// TIA Portal V20 export
// export: Created 2025-12-01T14:56:18.2640072Z, ExportSetting None, DisplayName Totally Integrated Automation Portal, DisplayVersion V20 Update 3, DisplayName TIA Portal Openness, DisplayVersion V20 Update 3, DisplayName TIA Portal Version Control Interface, DisplayVersion V20 Update 3, DisplayName STEP 7 Professional, DisplayVersion V20 Update 3, DisplayName STEP 7 Safety, DisplayVersion V20 Update 2, DisplayName WinCC Basic/Comfort/Advanced, DisplayVersion V20 Update 3, DisplayName WinCC Professional, DisplayVersion V20 Update 3, DisplayName WinCC Unified, DisplayVersion V20 Update 3
TYPE "UDT_VarLenze"
   STRUCT
      VF_Aviso : Bool;
      VF_Problema : Bool;
      VF01_EnAvance : Bool;
      VF01_EnRetroceso : Bool;
      VF02_EnAvance : Bool;
      VF02_EnRetroceso : Bool;
      VF01_Orden : Bool;
      VF02_Orden : Bool;
      VF_Ready : Bool;
      VF_SpeedCero : Bool;
      VF_NodoPresente : Bool;
      Bit_13 : Bool;
      Bit_14 : Bool;
      Bit_15 : Bool;
      Bit_16 : Bool;
      VF_SalidaDigital : Bool;
      ConsignaReal : Int;
      ConsignaReal_TMP : DInt;
      TIMConMutacion : UDInt;   // Temporizador de ConMutación de los Motores
   END_STRUCT;
END_TYPE
